# EPICS autosave request: iocBoot/iocsri/auto_settings.req
file sri_settings.req P=$(P)
